SUBAPPLICATION Ventilsteuerung_Uebung_072c (* GBSD auf UT ausgeben *)
  (* Standard: 61499-2 *)
  (* Version 1.0, 2023-10-23, franz *)
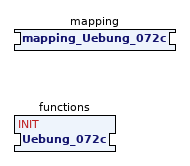
  SUBAPPS
    mapping : mapping_Uebung_072c;
    functions : Uebung_072c;
  END_SUBAPPS
END_SUBAPPLICATION
